// TIA Portal project "siemensxpython" (V16)

(* hardware
DEVICE "Station S7300/ET200M_1"  S7-300 station
   slot 0: "Châssis_0"  Rail  6ES7 390-1***0-0AA0
   slot 2: "PLC_1"  CPU 315-2 DP  6ES7 315-2AH14-0AB0  V3.3
      slot 0: "Interface MPI_1"  MPI
      slot 1: "Interface DP_1"  DP
   slot 4: "CP 343-1 Lean_1"  CP 343-1 LEAN  6GK7 343-1CX10-0XE0  V3.0
   slot 6: "DO 32x24VDC/0.5A_1"  DO32 x 24VDC / 0.5A  6ES7 322-1BL00-0AA0
*)

// ===== PLC "PLC_1"  CPU 315-2 DP =====

VAR_GLOBAL   // PLC tag table "Table de variables standard"
   "Tag_7" AT %Q0.0 : Bool;
   "Tag_8" AT %Q0.1 : Bool;
   "Tag_9" AT %Q0.2 : Bool;
   "Tag_10" AT %Q0.3 : Bool;
   "Tag_11" AT %Q0.4 : Bool;
   "Tag_12" AT %Q0.5 : Bool;
   "Tag_13" AT %Q0.6 : Bool;
   "Tag_14" AT %Q0.7 : Bool;
   "Tag_15" AT %Q1.1 : Bool;
   "Tag_16" AT %Q1.2 : Bool;
   "Tag_17" AT %Q1.0 : Bool;
   "Tag_18" AT %Q1.3 : Bool;
   "Tag_19" AT %Q1.4 : Bool;
   "Tag_20" AT %Q1.5 : Bool;
   "Tag_21" AT %Q1.6 : Bool;
   "Tag_22" AT %Q2.0 : Bool;
   "Tag_23" AT %Q2.1 : Bool;
   "Tag_24" AT %Q2.2 : Bool;
   "Tag_25" AT %Q2.3 : Bool;
   "Tag_26" AT %Q2.4 : Bool;
   "Tag_27" AT %Q2.5 : Bool;
   "Tag_28" AT %Q2.6 : Bool;
   "Tag_29" AT %Q2.7 : Bool;
   "Tag_30" AT %Q3.0 : Bool;
   "Tag_31" AT %Q3.1 : Bool;
   "Tag_32" AT %Q3.2 : Bool;
   "Tag_33" AT %Q3.3 : Bool;
   "Tag_34" AT %Q3.4 : Bool;
   "Tag_35" AT %Q3.5 : Bool;
   "Tag_36" AT %Q3.6 : Bool;
   "Tag_37" AT %Q3.7 : Bool;
   "Tag_38" AT %Q1.7 : Bool;
END_VAR

DATA_BLOCK "DB_python"   // DB1
{ S7_Optimized_Access := 'FALSE' }
VERSION : 0.1
   VAR
      S1 : Bool;
      S2 : Bool;
      S3 : Bool;
      S4 : Bool;
      S5 : Bool;
      S6 : Bool;
      S7 : Bool;
      S8 : Bool;
      S9 : Bool;
      S10 : Bool;
      S11 : Bool;
      S12 : Bool;
      S13 : Bool;
      S14 : Bool;
      S15 : Bool;
      S16 : Bool;
      S17 : Bool;
      S18 : Bool;
      S19 : Bool;
      S20 : Bool;
      S21 : Bool;
      S22 : Bool;
      S23 : Bool;
      S24 : Bool;
      S25 : Bool;
      S26 : Bool;
      S27 : Bool;
      S28 : Bool;
      S29 : Bool;
      S30 : Bool;
      S31 : Bool;
      S32 : Bool;
   END_VAR
BEGIN
END_DATA_BLOCK

ORGANIZATION_BLOCK "Main"   // OB1, LAD
TITLE = "Main Program Sweep (Cycle)"
{ S7_Optimized_Access := 'FALSE' }
VERSION : 0.1
   VAR_TEMP
      OB1_EV_CLASS : Byte;   // Bits 0-3 = 1 (Coming event), Bits 4-7 = 1 (Event class 1)
      OB1_SCAN_1 : Byte;   // 1 (Cold restart scan 1 of OB 1), 3 (Scan 2-n of OB 1)
      OB1_PRIORITY : Byte;   // Priority of OB Execution
      OB1_OB_NUMBR : Byte;   // 1 (Organization block 1, OB1)
      OB1_RESERVED_1 : Byte;   // Reserved for system
      OB1_RESERVED_2 : Byte;   // Reserved for system
      OB1_PREV_CYCLE : Int;   // Cycle time of previous OB1 scan (milliseconds)
      OB1_MIN_CYCLE : Int;   // Minimum cycle time of OB1 (milliseconds)
      OB1_MAX_CYCLE : Int;   // Maximum cycle time of OB1 (milliseconds)
      OB1_DATE_TIME : Date_And_Time;   // Date and time OB1 started
   END_VAR
BEGIN
END_ORGANIZATION_BLOCK